// TIA Portal V20 export
TYPE "LBP_typeModularMcpKeypadRecord"
TITLE = Modular MCP image / Image MCP modulaire
// Image of modular MCP for key properties / Image des MCP modulaires pour propriétés des touches
   STRUCT
      recordVersion : Byte := 16#10;   // version 1.0
      keyActiveAttributesCount : USInt;   // number of valid entries in keyActiveAttributes / nombre d'entrées valides dans keyActiveAttributes
      keyInactiveAttributesCount : USInt;   // number of valid entries in keyInactiveAttributes / nombre d'entrées valides dans keyInactiveAttributes
      reserved : Byte;   // unused variable / variable inutilisée
      keyActiveAttributes { S7_SetPoint := 'True'} : Array[0..20] of "LBP_typeModularMcpLedAttribute";   // color attributes for keys in state "active" / attributs de couleur pour les touches à l'état "actif"
      keyInactiveAttributes { S7_SetPoint := 'True'} : Array[0..20] of "LBP_typeModularMcpLedAttribute";   // color attributes for keys in state "inactive" / attributs de couleur pour les touches à l'état "inactif"
   END_STRUCT;
END_TYPE
